// TIA Portal project "IMPROVED_PROGRAM" (V16)

(* hardware
DEVICE "S7-1200 station_1"  S7-1200 Station
   slot 0: "Rack_0"  S7-1200 Rack  Rack  V1.0
   slot 1: "PLC_1"  CPU 1214C DC/DC/DC  6ES7 214-1AG40-0XB0  V4.4
DEVICE "SINAMICS G_1"  Sinamics.Device
   slot 0: "	_0"  Rail  SinamicsG120SVecto
   slot 0: "Drive_1"  G120 CU250S-2 PN Vector  6SL3246-0BA22-1FA0  4.7.10
      slot 1: "PROFINET interface"  MDD-SinamicsG120-P
   slot 3: "PM240-2 IP20"  PM240-2 IP20  6SL3210-1PB13-8ULx  -
DEVICE "ktp700"  KTP700 Basic PN
   slot 0: "ktp700"  KTP700 Basic PN  6AV2 123-2GB03-0AX0  16.0.0.0
   slot 1: "HMI_RT_1"  KTP700 Basic PN  6AV2 123-2GB03-0AX0  16.0.0.0
   slot 5: "ktp700.IE_CP_1"  PROFINET Interface  16.0.0.0
      slot 1: "PROFINET Interface_1"  PROFINET Interface
         slot 1: "Port_1"  Port
*)

// ===== PLC "PLC_1"  CPU 1214C DC/DC/DC =====

VAR_GLOBAL   // PLC tag table "Default tag table"
   "FORWARD" AT %I0.0 : Bool;
   "STOP" AT %I0.2 : Bool;
   "REVERSE" AT %I0.1 : Bool;
   "FLOOR_1_LS" AT %I0.5 : Bool;
   "FLOOR_2_LS" AT %I0.4 : Bool;
   "FLOOR_3_LS" AT %I0.3 : Bool;
   "SPEED" AT %MD1 : Real;
   "HMI_1ST_FLOOR" AT %M0.5 : Bool;
   "HMI_2ND_FLOOR" AT %M0.6 : Bool;
   "HMI_3RD_FLOOR" AT %M0.7 : Bool;
   "HMI_STOP" AT %M5.2 : Bool;
   "HMI_FLOOR_INDICATOR" AT %M5.3 : Bool;
   "Display_current" AT %MD18 : Real;
   "Display_torque" AT %MD22 : Real;
   "CONTROL" AT %ID15 : Real;
END_VAR

VAR_GLOBAL   // PLC tag table "unity"
   "ON/OFF_MEM" AT %M0.0 : Bool;
   "DIRECTION_MEM" AT %M0.1 : Bool;
   "FLOOR_MEM" AT %M0.2 : Bool;
   "FORWARD_MEM" AT %M0.3 : Bool;
   "REVERSE_MEM" AT %M0.4 : Bool;
   "START_MEM" AT %M5.0 : Bool;
   "STOP_MEM" AT %M5.1 : Bool;
   "CURRENT_FLOOR" AT %MD10 : DWord;
   "FLOOR_3_LS_MEM" AT %M5.5 : Bool;
   "FLOOR_2_LS_MEM" AT %M5.6 : Bool;
   "FLOOR_1_LS_MEM" AT %M5.4 : Bool;
   "Display_speed" AT %MD14 : Real;
   "Tag_1" AT %M6.0 : Bool;
   "Tag_4" AT %MD12 : Real;
   "Tag_2" AT %MD7 : Real;
   "Tag_3" AT %MD8 : Real;
   "Tag_5" AT %MD16 : DWord;
END_VAR

DATA_BLOCK "PZD_G120_Tel_352 V14_DB"   // DB1
{ S7_Optimized_Access := 'FALSE' }
VERSION : 0.1
// stored: InstanceOfName PZD_G120_Tel_352 V14
"PZD_G120_Tel_352 V14"
BEGIN
END_DATA_BLOCK

// folder: System blocks/Program resources

DATA_BLOCK "FLOOR_TIMER_NEW"   // DB2
{ S7_Optimized_Access := 'TRUE' }
AUTHOR : Simatic
FAMILY : IEC
NAME : IEC_TMR
VERSION : 1.0
// stored: InstanceOfName IEC_TIMER
"IEC_TIMER"
BEGIN
END_DATA_BLOCK

// folder: (top level)

FUNCTION_BLOCK "PZD_G120_Tel_352 V14"   // FB10, SCL
{ S7_Optimized_Access := 'FALSE' }
VERSION : 0.1
// PZD_G120_Tel_352
   VAR_INPUT
      address : Hw_Io := 0;   // I/O address of SINAMICS G120
      ON_OFF1 : Bool := FALSE;   // Bit 0: 0=OFF; 1=ON
      OFF2 : Bool := TRUE;   // Bit 1: 0=immediately STOP
      OFF3 : Bool := TRUE;   // Bit 2: 0=quick STOP
      enable_operation : Bool := TRUE;   // Bit 3: 0=cancel pulses
      release_RFG : Bool := TRUE;   // Bit 4: 0= RFG is set to 0; 1=RFG follows setpoint
      enable_RFG : Bool := TRUE;   // Bit 5: 0= freeze RFG, 1= 1=RFG follows setpoint
      enable_setpoint : Bool := TRUE;   // Bit 6: 0= setpoint is 0; 1=setpoint enabled
      acknowledge : Bool := FALSE;   // Bit 7: 0 to 1 = fault acknowledge
      CTW_bit_08 : Bool := FALSE;   // Bit 8: not used
      CTW_bit_09 : Bool := FALSE;   // Bit 9: not used
      PLC_is_master : Bool := TRUE;   // Bit10: 1= PLC controls the drive
      direction_reversal : Bool := FALSE;   // Bit11: 1= reverse turning direction
      CTW_bit_12 : Bool := FALSE;   // Bit12: not used
      MOP_up : Bool := FALSE;   // Bit13: increase setpoint in motorized Potentiometer
      MOP_down : Bool := FALSE;   // Bit14: decrease setpoint in motorized Potentiometer
      CTW_bit_15 : Bool := FALSE;   // Bit15: not used
      activate_manual_mode : Bool := FALSE;   // 0=Normal Mode; 1= Manual Mode (FB internal CTW and Setpoint)
      speed_setpoint : Real := 0.0;   // speed setpoint in turns/min
      reference_speed_P2000 : Real := 1500.0;   // reference value for speed, stored in P2000 ot the SINAMICS
      reference_current_P2002 : Real := 0.0;   // reference value for current, stored in P2002 ot the SINAMICS G120
      reference_torque_P2003 : Real := 0.0;   // reference value for torque, stored in P2003 ot the SINAMICS G120
   END_VAR
   VAR_OUTPUT
      ready_for_switching_on : Bool;   // Power supply is on, pulses are blocked
      ready_for_operation : Bool;   // Motor is switched on
      operation_enabled : Bool;   // Motor follows setpoint
      fault_active : Bool;   // SINAMICS shows a fault/error
      OFF2_inactive : Bool;   // No immediately STOP
      OFF3_inactive : Bool;   // No quick STOP
      closing_lockout_active : Bool;   // Switch on is inhibit, ON_OFF1 must be set to 0
      alarm_active : Bool;   // SINAMICS shows a alarm/warning
      speed_deviation_in_tol : Bool;   // Setpoint/actual value deviation within tolerance range.
      PLC_control_requested : Bool;   // PLC is requested to assume control
      comp_speed_reached : Bool;   // Speed is greater than or equal to the corresponding maximum speed.
      limit_reached : Bool;   // Comparison value for current, torque or power has been reached or exceeded.
      holding_brake_open : Bool;   // Signal to open and close a motor holding brake.
      alarm_motor_overtemp : Bool;   // Alarm motor overtemperature
      rotating_right : Bool;   // Internal inverter actual value > 0
      no_thermal_overload : Bool;   // No alarm, thermal power unit overload
      actual_speed : Real;   // actual speed of motot in turns/min
      actual_current : Real;   // actual current in A
      actual_torque : Real;   // actual torque in Nm
      actual_alarm : Word;   // actual alarm/warning
      actual_fault : Word;   // actual fault/error
   END_VAR
   VAR
      internal_control_word : Word := W#16#047E;   // control word for manual mode
      internal_status_word : Word := 16#0000;   // status word for manual mode
      internal_setpoint : Real := 0.0;   // setpoint for manual mode
      return_value_RD : Int := 0;   // return value from SFC 14
      return_value_WR : Int := 0;   // return value from SFC 15
      ValueMax : Real := 16384.0;
      InData : Array[1..12] of Byte;   // received data
      InData_word AT InData : Array[1..6] of Word;
      OutData : Array[1..12] of Byte;   // data to send
      OutData_word AT OutData : Array[1..6] of Word;
   END_VAR
   VAR_TEMP
      Control_word : Word;   // control word for drive
      Control_word_bits AT Control_word : Struct
         Bit_00 : Bool;
         Bit_01 : Bool;
         Bit_02 : Bool;
         Bit_03 : Bool;
         Bit_04 : Bool;
         Bit_05 : Bool;
         Bit_06 : Bool;
         Bit_07 : Bool;
         Bit_08 : Bool;
         Bit_09 : Bool;
         Bit_10 : Bool;
         Bit_11 : Bool;
         Bit_12 : Bool;
         Bit_13 : Bool;
         Bit_14 : Bool;
         Bit_15 : Bool;
      END_STRUCT;
      Status_word : Word;   // status word for drive
      Status_word_bits AT Status_word : Struct   // bits of the status word
         Bit_00 : Bool;
         Bit_01 : Bool;
         Bit_02 : Bool;
         Bit_03 : Bool;
         Bit_04 : Bool;
         Bit_05 : Bool;
         Bit_06 : Bool;
         Bit_07 : Bool;
         Bit_08 : Bool;
         Bit_09 : Bool;
         Bit_10 : Bool;
         Bit_11 : Bool;
         Bit_12 : Bool;
         Bit_13 : Bool;
         Bit_14 : Bool;
         Bit_15 : Bool;
      END_STRUCT;
      tempout_int : Int;
      tempout_real : Real;
   END_VAR
BEGIN
   //RECEIVE DATA
   //Copy all 6 received words (Siemens telegram 352) to buffer (with SFC14 DPRD_DAT)
   #return_value_RD := DPRD_DAT(LADDR := #address,RECORD => #InData);

   //CONVERT STATUS WORD AND COPY TO OUTPUTS
   //The SINAMICS and the SIMATIC uses different Byte orders (Endianness)
   //The SINAMICS use Intel format or Little-Endian while the SIMATIC uses Motorola format or Big-Endian.
   //The control and status words have to be change the high AND low bytes.
   #Status_word :=  ROL(IN:=#InData_word[1] ,N:=8);
   #internal_status_word := #InData_word[1];

   //copy bits of the status word to output
   #ready_for_switching_on      := #Status_word_bits.Bit_00 ;//Power supply is on, pulses are blocked
   #ready_for_operation         := #Status_word_bits.Bit_01 ;//Motor is switched on
   #operation_enabled           := #Status_word_bits.Bit_02 ;//Motor follows setpoint
   #fault_active                := #Status_word_bits.Bit_03 ;//SINAMICS shows a fault/error
   #OFF2_inactive               := #Status_word_bits.Bit_04 ;//No immediately STOP
   #OFF3_inactive               := #Status_word_bits.Bit_05 ;//No quick STOP
   #closing_lockout_active      := #Status_word_bits.Bit_06 ;//Switch on is inhibit, ON_OFF1 must be set to 0
   #alarm_active                := #Status_word_bits.Bit_07 ;//SINAMICS shows a alarm/warning
   #speed_deviation_in_tol      := #Status_word_bits.Bit_08 ;//Setpoint/actual value deviation within tolerance range. 
   #PLC_control_requested       := #Status_word_bits.Bit_09 ;//PLC is requested to assume control
   #comp_speed_reached          := #Status_word_bits.Bit_10 ;//Speed is greater than or equal to the corresponding maximum speed.
   #limit_reached               := #Status_word_bits.Bit_11 ;//Comparison value for current, torque or power has been reached or exceeded.
   #holding_brake_open          := #Status_word_bits.Bit_12 ;//Signal to open and close a motor holding brake.
   #alarm_motor_overtemp        := #Status_word_bits.Bit_13 ;//Alarm motor overtemperature
   #rotating_right              := #Status_word_bits.Bit_14 ;//Internal inverter actual value > 0 
   #no_thermal_overload         := #Status_word_bits.Bit_15 ;//No alarm, thermal power unit overload

   //CONVERT ACTUAL VALUES AND COPY TO OUTPUTS
   //The speed, current and torque values are transferred as scaled values.
   //The reference speed for the scaling is stored in P2000 in a SINAMICS G120. 
   //The reference current for the scaling is stored in P2002 in a SINAMICS G120. 
   //The reference torque for the scaling is stored in P2003 in a SINAMICS G120. 
   //The scaling is: 100%(of P200x)=4000hex=16384dez  

   #actual_speed   := #reference_speed_P2000   * ( INT_TO_REAL( WORD_TO_INT(#InData_word[2])) / #ValueMax );
   #actual_current := #reference_current_P2002 * ( INT_TO_REAL( WORD_TO_INT(#InData_word[3])) / #ValueMax );
   #actual_torque  := #reference_torque_P2003  * ( INT_TO_REAL( WORD_TO_INT(#InData_word[4])) / #ValueMax );

   //COPY ALARM/FAULT CODES TO OUTPUTS
   #actual_alarm := #InData_word[5] ;   
   #actual_fault := #InData_word[6] ;  

   // ###########################################

   // Depending on activate_manual_mode we copy the input variables or the internen variables to the output buffer
   IF #activate_manual_mode = FALSE THEN // normal mode
       //COPY INPUT BITS
       #Control_word_bits.Bit_00 := #ON_OFF1;            //Bit 0: 0=immediately STOP
       #Control_word_bits.Bit_01 := #OFF2;               //Bit 1: 0=cancel pulses
       #Control_word_bits.Bit_02 := #OFF3;               //Bit 2: 0=quick STOP
       #Control_word_bits.Bit_03 := #enable_operation;   //Bit 3: 0=cancel pulses

       #Control_word_bits.Bit_04 := #enable_RFG;         //Bit 4: 0= setpoint is 0; 1=setpoint enabled
       #Control_word_bits.Bit_05 := #enable_setpoint;    //Bit 5: 0= freeze RFG, 1= 1=RFG follows setpoint
       #Control_word_bits.Bit_06 := #enable_setpoint;    //Bit 6: 1= enable setpoint
       #Control_word_bits.Bit_07 := #acknowledge;        //Bit 7: 0 to 1 = fault acknowledge

       #Control_word_bits.Bit_08 := #CTW_bit_08;         //Bit 8: not used
       #Control_word_bits.Bit_09 := #CTW_bit_09;         //Bit 9: not used
       #Control_word_bits.Bit_10 := #PLC_is_master;      //Bit10: 1= PLC controls the drive
       #Control_word_bits.Bit_11 := #direction_reversal; //Bit11: 1= reverse turning direction

       #Control_word_bits.Bit_12 := #CTW_bit_12;         //Bit12: not used
       #Control_word_bits.Bit_13 := #MOP_up;             //Bit13: increase setpoint in motorized Potentiometer
       #Control_word_bits.Bit_14 := #MOP_down;           //Bit14: decrease setpoint in motorized Potentiometer
       #Control_word_bits.Bit_15 := #CTW_bit_15;         //Bit15: not used

       //CONVERT AND COPY CONTROL WORD TO BUFFER
       //The SINAMICS and the SIMATIC uses different Byte orders (Endianness)
       //The SINAMICS use Intel format or Little-Endian while the SIMATIC uses Motorola format or Big-Endian.
       //The control and status words have to be change the high AND low bytes.
       #OutData_word[1] :=  ROL(IN:=#Control_word ,N:=8);

       //CONVERT SETPOINT VALUE AND COPY TO BUFFER
       //The speed value is transferred as scaled value.
       //The reference speed for the scaling is stored in P2000 in a SINAMICS G120. 
       //The scaling is: 100%(of P2000)=4000hex=16384dez  
       #OutData_word[2]:=INT_TO_WORD (REAL_TO_INT (#speed_setpoint * #ValueMax / #reference_speed_P2000));

   ELSE    //manual mode
       //CONVERT AND COPY CONTROL WORD TO BUFFER
       //The SINAMICS and the SIMATIC uses different Byte orders (Endianness)
       //The SINAMICS use Intel format or Little-Endian while the SIMATIC uses Motorola format or Big-Endian.
       //The control and status words have to be change the high AND low bytes.
       #OutData_word[1] :=  #internal_control_word;

       //CONVERT SETPOINT VALUE AND COPY TO BUFFER
       //The speed value is transferred as scaled value.
       //The reference speed for the scaling is stored in P2000 in a SINAMICS G120. 
       //The scaling is: 100%(of P2000)=4000hex=16384dez  
       #OutData_word[2]:=INT_TO_WORD (REAL_TO_INT (#internal_setpoint * #ValueMax / #reference_speed_P2000));
   END_IF;

   //FILL NOT USED WORDS IN BUFFER
   #OutData_word[3]:= INT_TO_WORD (0);
   #OutData_word[4]:= INT_TO_WORD (0);
   #OutData_word[5]:= INT_TO_WORD (0);
   #OutData_word[6]:= INT_TO_WORD (0);

   //SEND DATA
   //Copy all 6 words (Siemens telegram 352) from buffer (with SFC15 DPWR_DAT)
   #return_value_WR := DPWR_DAT(LADDR := #address,RECORD := #OutData );
END_FUNCTION_BLOCK

ORGANIZATION_BLOCK "Main"   // OB1, LAD, ProgramCycle
TITLE = "ELEVATOR_CONTROL_LOGIC"
{ S7_Optimized_Access := 'TRUE' }
VERSION : 0.1
   VAR_INPUT
      Initial_Call : Bool;   // Initial call of this OB
      Remanence : Bool;   // =True, if remanent data are available
   END_VAR
BEGIN

REGION Network 1: VFD_DRIVE_BLOCK
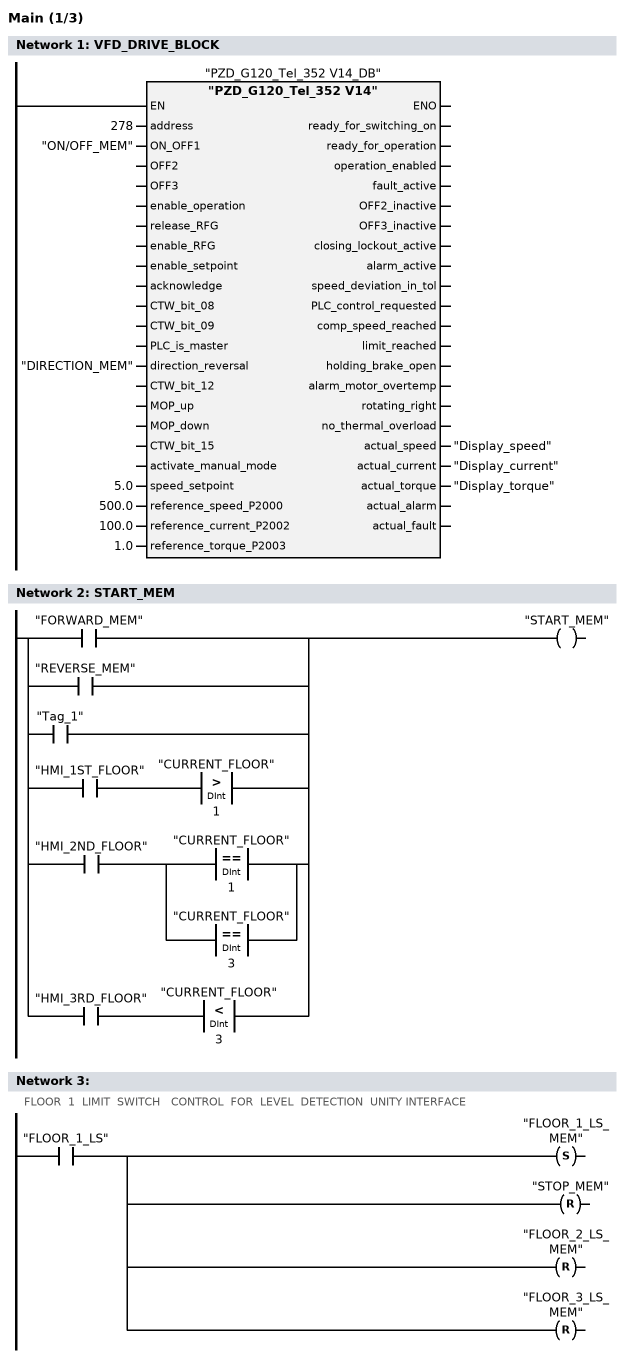
   RUNG wire#powerrail
      "PZD_G120_Tel_352 V14_DB"(address := 278, ON_OFF1 := "ON/OFF_MEM", OFF2 :=, OFF3 :=, enable_operation :=, release_RFG :=, enable_RFG :=, enable_setpoint :=, acknowledge :=, CTW_bit_08 :=, CTW_bit_09 :=, PLC_is_master :=, direction_reversal := "DIRECTION_MEM", CTW_bit_12 :=, MOP_up :=, MOP_down :=, CTW_bit_15 :=, activate_manual_mode :=, speed_setpoint := 5.0, reference_speed_P2000 := 500.0, reference_current_P2002 := 100.0, reference_torque_P2003 := 1.0, ready_for_switching_on =>, ready_for_operation =>, operation_enabled =>, fault_active =>, OFF2_inactive =>, OFF3_inactive =>, closing_lockout_active =>, alarm_active =>, speed_deviation_in_tol =>, PLC_control_requested =>, comp_speed_reached =>, limit_reached =>, holding_brake_open =>, alarm_motor_overtemp =>, rotating_right =>, no_thermal_overload =>, actual_speed => "Display_speed", actual_current => "Display_current", actual_torque => "Display_torque", actual_alarm =>, actual_fault =>)
   END_RUNG
   // the same network as SCL:
   "PZD_G120_Tel_352 V14_DB"(address := 278,   // "PZD_G120_Tel_352 V14"
                           ON_OFF1 := "ON/OFF_MEM",
                           direction_reversal := "DIRECTION_MEM",
                           speed_setpoint := 5.0,
                           reference_speed_P2000 := 500.0,
                           reference_current_P2002 := 100.0,
                           reference_torque_P2003 := 1.0,
                           actual_speed => "Display_speed",
                           actual_current => "Display_current",
                           actual_torque => "Display_torque");
END_REGION

REGION Network 2: START_MEM
   RUNG wire#powerrail
      Contact( "FORWARD_MEM" )
      wire#w1
      Coil( "START_MEM" )
   END_RUNG
   RUNG wire#powerrail
      Contact( "REVERSE_MEM" )
   END_RUNG wire#w1
   RUNG wire#powerrail
      Contact( "Tag_1" )
   END_RUNG wire#w1
   RUNG wire#powerrail
      Contact( "HMI_1ST_FLOOR" )
      { S7_Templates := "SrcType := DInt" } GT_Contact(in1 := "CURRENT_FLOOR", in2 := 1)
   END_RUNG wire#w1
   RUNG wire#powerrail
      Contact( "HMI_2ND_FLOOR" )
      wire#w2
      { S7_Templates := "SrcType := DInt" } EQ_Contact(in1 := "CURRENT_FLOOR", in2 := 1)
   END_RUNG wire#w1
   RUNG wire#w2
      { S7_Templates := "SrcType := DInt" } EQ_Contact(in1 := "CURRENT_FLOOR", in2 := 3)
   END_RUNG wire#w1
   RUNG wire#powerrail
      Contact( "HMI_3RD_FLOOR" )
      { S7_Templates := "SrcType := DInt" } LT_Contact(in1 := "CURRENT_FLOOR", in2 := 3)
   END_RUNG wire#w1
   // the same network as SCL:
   "START_MEM" := "FORWARD_MEM" OR "REVERSE_MEM" OR "Tag_1" OR ("HMI_1ST_FLOOR" AND ("CURRENT_FLOOR" > 1)) OR ("HMI_2ND_FLOOR" AND (("CURRENT_FLOOR" = 1) OR ("CURRENT_FLOOR" = 3))) OR ("HMI_3RD_FLOOR" AND ("CURRENT_FLOOR" < 3));
END_REGION

REGION Network 3
   // FLOOR  1  LIMIT  SWITCH   CONTROL  FOR  LEVEL  DETECTION  UNITY INTERFACE
   RUNG wire#powerrail
      Contact( "FLOOR_1_LS" )
      wire#w1
      S_Coil( "FLOOR_1_LS_MEM" )
   END_RUNG
   RUNG wire#w1
      R_Coil( "STOP_MEM" )
   END_RUNG
   RUNG wire#w1
      R_Coil( "FLOOR_2_LS_MEM" )
   END_RUNG
   RUNG wire#w1
      R_Coil( "FLOOR_3_LS_MEM" )
   END_RUNG
   // the same network as SCL:
   IF "FLOOR_1_LS" THEN
       "FLOOR_1_LS_MEM" := TRUE;
       "STOP_MEM" := FALSE;
       "FLOOR_2_LS_MEM" := FALSE;
       "FLOOR_3_LS_MEM" := FALSE;
   END_IF;
END_REGION

REGION Network 4
   // FLOOR  TWO  LIMIT  SWITCH  DETECTION  AND  CONTROL   UNITY  INTERFACE
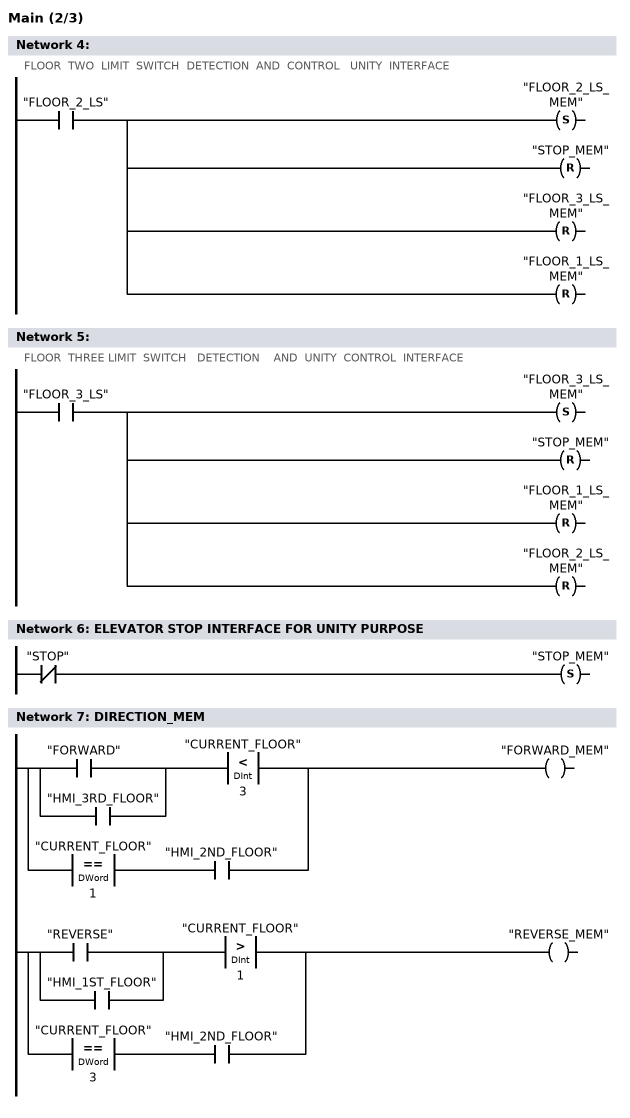
   RUNG wire#powerrail
      Contact( "FLOOR_2_LS" )
      wire#w1
      S_Coil( "FLOOR_2_LS_MEM" )
   END_RUNG
   RUNG wire#w1
      R_Coil( "STOP_MEM" )
   END_RUNG
   RUNG wire#w1
      R_Coil( "FLOOR_3_LS_MEM" )
   END_RUNG
   RUNG wire#w1
      R_Coil( "FLOOR_1_LS_MEM" )
   END_RUNG
   // the same network as SCL:
   IF "FLOOR_2_LS" THEN
       "FLOOR_2_LS_MEM" := TRUE;
       "STOP_MEM" := FALSE;
       "FLOOR_3_LS_MEM" := FALSE;
       "FLOOR_1_LS_MEM" := FALSE;
   END_IF;
END_REGION

REGION Network 5
   // FLOOR  THREE LIMIT  SWITCH   DETECTION    AND  UNITY  CONTROL  INTERFACE
   RUNG wire#powerrail
      Contact( "FLOOR_3_LS" )
      wire#w1
      S_Coil( "FLOOR_3_LS_MEM" )
   END_RUNG
   RUNG wire#w1
      R_Coil( "STOP_MEM" )
   END_RUNG
   RUNG wire#w1
      R_Coil( "FLOOR_1_LS_MEM" )
   END_RUNG
   RUNG wire#w1
      R_Coil( "FLOOR_2_LS_MEM" )
   END_RUNG
   // the same network as SCL:
   IF "FLOOR_3_LS" THEN
       "FLOOR_3_LS_MEM" := TRUE;
       "STOP_MEM" := FALSE;
       "FLOOR_1_LS_MEM" := FALSE;
       "FLOOR_2_LS_MEM" := FALSE;
   END_IF;
END_REGION

REGION Network 6: ELEVATOR STOP INTERFACE FOR UNITY PURPOSE
   RUNG wire#powerrail
      I_Contact( "STOP" )
      S_Coil( "STOP_MEM" )
   END_RUNG
   // the same network as SCL:
   IF NOT "STOP" THEN "STOP_MEM" := TRUE; END_IF;
END_REGION

REGION Network 7: DIRECTION_MEM
   RUNG wire#powerrail
      Contact( "FORWARD" )
      wire#w1
      { S7_Templates := "SrcType := DInt" } LT_Contact(in1 := "CURRENT_FLOOR", in2 := 3)
      wire#w2
      Coil( "FORWARD_MEM" )
   END_RUNG
   RUNG wire#powerrail
      Contact( "HMI_3RD_FLOOR" )
   END_RUNG wire#w1
   RUNG wire#powerrail
      { S7_Templates := "SrcType := DWord" } EQ_Contact(in1 := "CURRENT_FLOOR", in2 := 1)
      Contact( "HMI_2ND_FLOOR" )
   END_RUNG wire#w2
   RUNG wire#powerrail
      Contact( "REVERSE" )
      wire#w3
      { S7_Templates := "SrcType := DInt" } GT_Contact(in1 := "CURRENT_FLOOR", in2 := 1)
      wire#w4
      Coil( "REVERSE_MEM" )
   END_RUNG
   RUNG wire#powerrail
      Contact( "HMI_1ST_FLOOR" )
   END_RUNG wire#w3
   RUNG wire#powerrail
      { S7_Templates := "SrcType := DWord" } EQ_Contact(in1 := "CURRENT_FLOOR", in2 := 3)
      Contact( "HMI_2ND_FLOOR" )
   END_RUNG wire#w4
   // the same network as SCL:
   "FORWARD_MEM" := (("FORWARD" OR "HMI_3RD_FLOOR") AND ("CURRENT_FLOOR" < 3)) OR (("CURRENT_FLOOR" = 1) AND "HMI_2ND_FLOOR");
   "REVERSE_MEM" := (("REVERSE" OR "HMI_1ST_FLOOR") AND ("CURRENT_FLOOR" > 1)) OR (("CURRENT_FLOOR" = 3) AND "HMI_2ND_FLOOR");
END_REGION

REGION Network 8: START_MOTOR
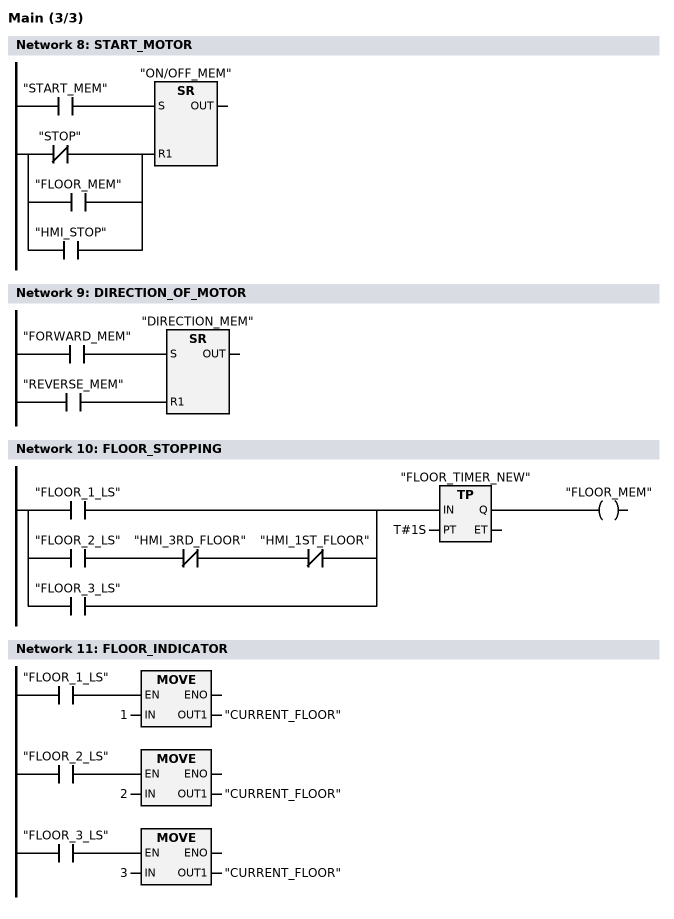
   RUNG wire#powerrail
      Contact( "START_MEM" )
      S_SR(operand := "ON/OFF_MEM", r1 := wire#w1)
   END_RUNG
   RUNG wire#powerrail
      I_Contact( "STOP" )
   END_RUNG wire#w1
   RUNG wire#powerrail
      Contact( "FLOOR_MEM" )
   END_RUNG wire#w1
   RUNG wire#powerrail
      Contact( "HMI_STOP" )
   END_RUNG wire#w1
   // the same network as SCL:
   IF "START_MEM" THEN
       "ON/OFF_MEM" := TRUE;   // SR flip-flop
   END_IF;
   IF NOT "STOP" OR "FLOOR_MEM" OR "HMI_STOP" THEN "ON/OFF_MEM" := FALSE; END_IF;
END_REGION

REGION Network 9: DIRECTION_OF_MOTOR
   RUNG wire#powerrail
      Contact( "FORWARD_MEM" )
      S_SR(operand := "DIRECTION_MEM", r1 := wire#w1)
   END_RUNG
   RUNG wire#powerrail
      Contact( "REVERSE_MEM" )
   END_RUNG wire#w1
   // the same network as SCL:
   IF "FORWARD_MEM" THEN
       "DIRECTION_MEM" := TRUE;   // SR flip-flop
   END_IF;
   IF "REVERSE_MEM" THEN "DIRECTION_MEM" := FALSE; END_IF;
END_REGION

REGION Network 10: FLOOR_STOPPING
   "FLOOR_TIMER_NEW".TP(IN := "FLOOR_1_LS" OR ("FLOOR_2_LS" AND NOT "HMI_3RD_FLOOR" AND NOT "HMI_1ST_FLOOR") OR "FLOOR_3_LS",
                        PT := T#1S);
   "FLOOR_MEM" := "FLOOR_TIMER_NEW".Q;
END_REGION

REGION Network 11: FLOOR_INDICATOR
   RUNG wire#powerrail
      Contact( "FLOOR_1_LS" )
      Move(in := 1, out1 => "CURRENT_FLOOR")
   END_RUNG
   RUNG wire#powerrail
      Contact( "FLOOR_2_LS" )
      Move(in := 2, out1 => "CURRENT_FLOOR")
   END_RUNG
   RUNG wire#powerrail
      Contact( "FLOOR_3_LS" )
      Move(in := 3, out1 => "CURRENT_FLOOR")
   END_RUNG
   // the same network as SCL:
   IF "FLOOR_1_LS" THEN "CURRENT_FLOOR" := 1; END_IF;
   IF "FLOOR_2_LS" THEN "CURRENT_FLOOR" := 2; END_IF;
   IF "FLOOR_3_LS" THEN "CURRENT_FLOOR" := 3; END_IF;
END_REGION
END_ORGANIZATION_BLOCK

ORGANIZATION_BLOCK "Cyclic interrupt"   // OB30, LAD, CyclicInterrupt
{ S7_Optimized_Access := 'TRUE' }
VERSION : 0.1
   VAR_INPUT
      Initial_Call : Bool;   // Initial call of this OB
      Event_Count : Int;   // Events discarded
   END_VAR
BEGIN

REGION Network 1
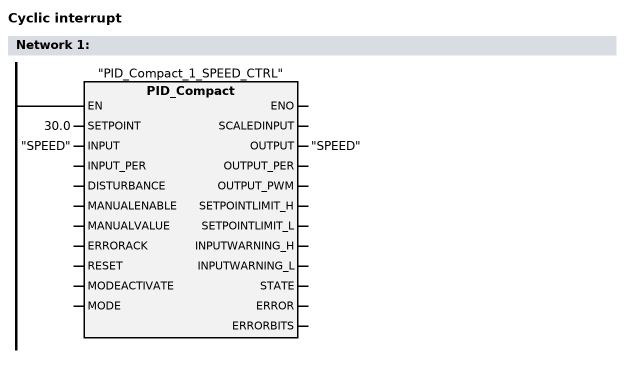
   "PID_Compact_1_SPEED_CTRL"(Setpoint := 30.0, Input := "SPEED", Output => "SPEED");   // PID_Compact
END_REGION
END_ORGANIZATION_BLOCK

(* ===== HMI "HMI_RT_1" =====
system functions are stored by id; their names below are inferred from use
connection "HMI_Connection_1": ETHERNET, SMART_S7_1200_OMS

HMI tags "Default tag table"
   "HMI_2ND_FLOOR" : Bool = PLC HMI_2ND_FLOOR AT %M0.6, 1 s
   "HMI_3RD_FLOOR" : Bool = PLC HMI_3RD_FLOOR AT %M0.7, 1 s
   "HMI_STOP" : Bool = PLC HMI_STOP AT %M5.2, 1 s
   "HMI_1ST_FLOOR" : Bool = PLC HMI_1ST_FLOOR AT %M0.5, 1 s
   "CURRENT_FLOOR" : DWord = PLC CURRENT_FLOOR AT %MD10, 1 s
   "HMI_Display_speed" : Real = PLC Display_speed AT %MD14, 1 s
   "HMI_Display_current" : Real = PLC Display_current AT %MD18, 1 s
   "HMI_Display_torque" : Real = PLC Display_torque AT %MD22, 1 s

screen "Screen_1" 800x480
   Button "Button_1" at 516,289 size 111x46; TextOff '1'
      on Press: SetBit("HMI_1ST_FLOOR"); ResetBit("HMI_2ND_FLOOR"); ResetBit("HMI_3RD_FLOOR"); ResetBit("HMI_STOP")
      Appearance <- "HMI_1ST_FLOOR"
   Button "Button_2" at 518,225 size 109x44; TextOff '2'
      on Press: SetBit("HMI_2ND_FLOOR"); ResetBit("HMI_1ST_FLOOR"); ResetBit("HMI_3RD_FLOOR"); ResetBit("HMI_STOP")
      Appearance <- "HMI_2ND_FLOOR"
   Button "Button_3" at 518,159 size 109x43; TextOff '3'
      on Press: SetBit("HMI_3RD_FLOOR"); ResetBit("HMI_1ST_FLOOR"); ResetBit("HMI_2ND_FLOOR"); ResetBit("HMI_STOP")
      Appearance <- "HMI_3RD_FLOOR"
   Button "Button_4" at 494,355 size 170x61; TextOff 'STOP'
      on Press: SetBit("HMI_STOP"); ResetBit("HMI_1ST_FLOOR"); ResetBit("HMI_2ND_FLOOR"); ResetBit("HMI_3RD_FLOOR")
      Appearance <- "HMI_STOP"
   IOField "I/O field_1" at 142,199 size 159x136; FormatPattern 9
      ProcessValue <- "CURRENT_FLOOR"
   TextField "Text field_1" at 143,175 size 136x27; Text 'FLOOR LEVEL'
   IOField "I/O field_2" at 20,74 size 107x46; FormatPattern 99.9; Unit  RPM
      ProcessValue <- "HMI_Display_speed"
   IOField "I/O field_3" at 154,74 size 90x46; FormatPattern 9.9; Unit  A
      ProcessValue <- "HMI_Display_current"
   IOField "I/O field_4" at 273,74 size 94x46; FormatPattern 99; Unit  Nm
      ProcessValue <- "HMI_Display_torque"
   TextField "Text field_2" at 24,51 size 64x23; Text 'SPEED:'
   TextField "Text field_3" at 154,50 size 91x23; Text 'CURRENT:'
   TextField "Text field_4" at 271,51 size 80x23; Text 'TORQUE:'
*)